PROGRAM PID_TempCtrl
VAR
	Heater10A_Temp_Reading_Raw		: INT;
	Stn10ActualTempRawData			: INT;
	Stn10HeaterRawData				: INT;

	STN10_PIDFB						: PID_FB;
	STN10_PIDCVFB					: DC_PID_FB;

	Stn10_PID_fKp					: REAL := 0.2					; (*1.0*)
	Stn10_PID_tTn					: TIME := T#1S				;
	Stn10_PID_tTv					: TIME := T#30MS				;
	Stn10_PID_tTd					: TIME := T#40MS				;



		iHeater10A_Temp_Output_Percent : INT;
END_VAR

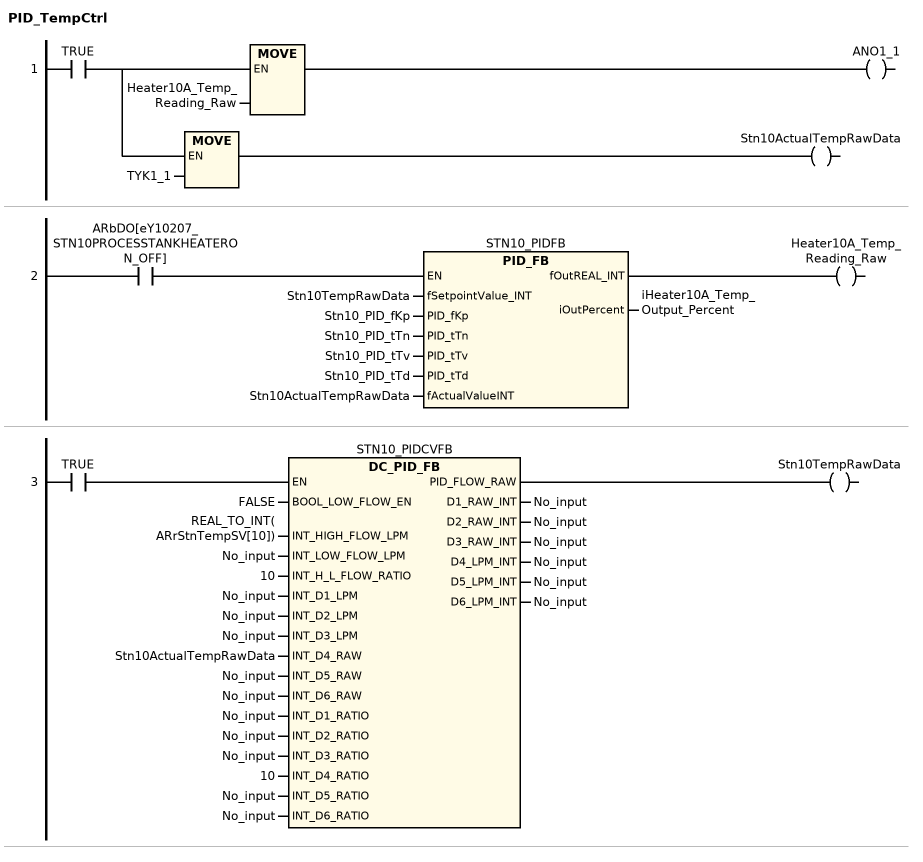
// NETWORK 1
ANO1_1 := Heater10A_Temp_Reading_Raw;
Stn10ActualTempRawData := TYK1_1;

// NETWORK 2
IF ARbDO[eY10207_STN10PROCESSTANKHEATERON_OFF] THEN
    STN10_PIDFB(
        fSetpointValue_INT := Stn10TempRawData,
        PID_fKp := Stn10_PID_fKp,
        PID_tTn := Stn10_PID_tTn,
        PID_tTv := Stn10_PID_tTv,
        PID_tTd := Stn10_PID_tTd,
        fActualValueINT := Stn10ActualTempRawData,
        iOutPercent => iHeater10A_Temp_Output_Percent); // PID_FB
END_IF
Heater10A_Temp_Reading_Raw := STN10_PIDFB.fOutREAL_INT;

// NETWORK 3
STN10_PIDCVFB(
    BOOL_LOW_FLOW_EN := FALSE,
    INT_HIGH_FLOW_LPM := REAL_TO_INT(ARrStnTempSV[10]),
    INT_LOW_FLOW_LPM := No_input,
    INT_H_L_FLOW_RATIO := 10,
    INT_D1_LPM := No_input,
    INT_D2_LPM := No_input,
    INT_D3_LPM := No_input,
    INT_D4_RAW := Stn10ActualTempRawData,
    INT_D5_RAW := No_input,
    INT_D6_RAW := No_input,
    INT_D1_RATIO := No_input,
    INT_D2_RATIO := No_input,
    INT_D3_RATIO := No_input,
    INT_D4_RATIO := 10,
    INT_D5_RATIO := No_input,
    INT_D6_RATIO := No_input,
    D1_RAW_INT => No_input,
    D2_RAW_INT => No_input,
    D3_RAW_INT => No_input,
    D4_LPM_INT => No_input,
    D5_LPM_INT => No_input,
    D6_LPM_INT => No_input); // DC_PID_FB
Stn10TempRawData := STN10_PIDCVFB.PID_FLOW_RAW;

END_PROGRAM

(* stored: Version 1.1.0.1, ProductVersion 3.1.4024.12
   POU PID_TempCtrl: Id {143dd274-7f18-46a1-9f8f-91015dfc0131}, SpecialFunc None *)
